// TIA Portal V18 export
FUNCTION "Deaering sequences" : Void   // FC4, LAD
{ S7_Optimized_Access := 'TRUE' }
VERSION : 0.1
// stored: AutoNumber true, IsIECCheckEnabled false, SetENOAutomatically false, UDAEnableTagReadback false
BEGIN

REGION Network 1: Dearing A with valve
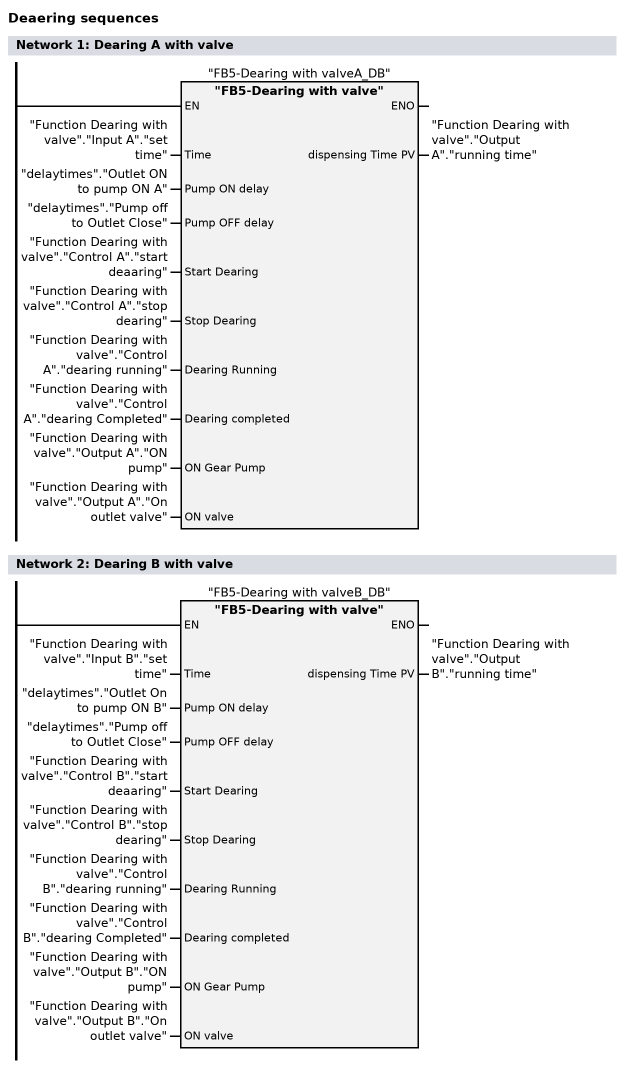
   RUNG wire#powerrail
      "FB5-Dearing with valveA_DB"("Time" := "Function Dearing with valve"."Input A"."set time", "Pump ON delay" := "delaytimes"."Outlet ON to pump ON A", "Pump OFF delay" := "delaytimes"."Pump off to Outlet Close", "Start Dearing" := "Function Dearing with valve"."Control A"."start deaaring", "Stop Dearing" := "Function Dearing with valve"."Control A"."stop dearing", "Dearing Running" := "Function Dearing with valve"."Control A"."dearing running", "Dearing completed" := "Function Dearing with valve"."Control A"."dearing Completed", "ON Gear Pump" := "Function Dearing with valve"."Output A"."ON pump", "ON valve" := "Function Dearing with valve"."Output A"."On outlet valve", "dispensing Time PV" => "Function Dearing with valve"."Output A"."running time")
   END_RUNG
   // the same network as SCL:
   "FB5-Dearing with valveA_DB"("Time" := "Function Dearing with valve"."Input A"."set time",   // "FB5-Dearing with valve"
                           "Pump ON delay" := "delaytimes"."Outlet ON to pump ON A",
                           "Pump OFF delay" := "delaytimes"."Pump off to Outlet Close",
                           "Start Dearing" := "Function Dearing with valve"."Control A"."start deaaring",
                           "Stop Dearing" := "Function Dearing with valve"."Control A"."stop dearing",
                           "Dearing Running" := "Function Dearing with valve"."Control A"."dearing running",
                           "Dearing completed" := "Function Dearing with valve"."Control A"."dearing Completed",
                           "ON Gear Pump" := "Function Dearing with valve"."Output A"."ON pump",
                           "ON valve" := "Function Dearing with valve"."Output A"."On outlet valve",
                           "dispensing Time PV" => "Function Dearing with valve"."Output A"."running time");
END_REGION

REGION Network 2: Dearing B with valve
   RUNG wire#powerrail
      "FB5-Dearing with valveB_DB"("Time" := "Function Dearing with valve"."Input B"."set time", "Pump ON delay" := "delaytimes"."Outlet On to pump ON B", "Pump OFF delay" := "delaytimes"."Pump off to Outlet Close", "Start Dearing" := "Function Dearing with valve"."Control B"."start deaaring", "Stop Dearing" := "Function Dearing with valve"."Control B"."stop dearing", "Dearing Running" := "Function Dearing with valve"."Control B"."dearing running", "Dearing completed" := "Function Dearing with valve"."Control B"."dearing Completed", "ON Gear Pump" := "Function Dearing with valve"."Output B"."ON pump", "ON valve" := "Function Dearing with valve"."Output B"."On outlet valve", "dispensing Time PV" => "Function Dearing with valve"."Output B"."running time")
   END_RUNG
   // the same network as SCL:
   "FB5-Dearing with valveB_DB"("Time" := "Function Dearing with valve"."Input B"."set time",   // "FB5-Dearing with valve"
                           "Pump ON delay" := "delaytimes"."Outlet On to pump ON B",
                           "Pump OFF delay" := "delaytimes"."Pump off to Outlet Close",
                           "Start Dearing" := "Function Dearing with valve"."Control B"."start deaaring",
                           "Stop Dearing" := "Function Dearing with valve"."Control B"."stop dearing",
                           "Dearing Running" := "Function Dearing with valve"."Control B"."dearing running",
                           "Dearing completed" := "Function Dearing with valve"."Control B"."dearing Completed",
                           "ON Gear Pump" := "Function Dearing with valve"."Output B"."ON pump",
                           "ON valve" := "Function Dearing with valve"."Output B"."On outlet valve",
                           "dispensing Time PV" => "Function Dearing with valve"."Output B"."running time");
END_REGION

REGION Network 3: Dearing A without Valve
END_REGION

REGION Network 4: Dearing B without Valve
END_REGION
END_FUNCTION
